// TIA Portal V18 export
ORGANIZATION_BLOCK "Main"   // OB1, LAD, ProgramCycle
TITLE = "Main Program Sweep (Cycle)"
{ S7_Optimized_Access := 'TRUE' }
VERSION : 0.1
// stored: AutoNumber true, IsIECCheckEnabled false, SetENOAutomatically false
   VAR_INPUT
      Initial_Call : Bool;   // Initial call of this OB
      Remanence : Bool;   // =True, if remanent data are available
   END_VAR
BEGIN

REGION Network 2
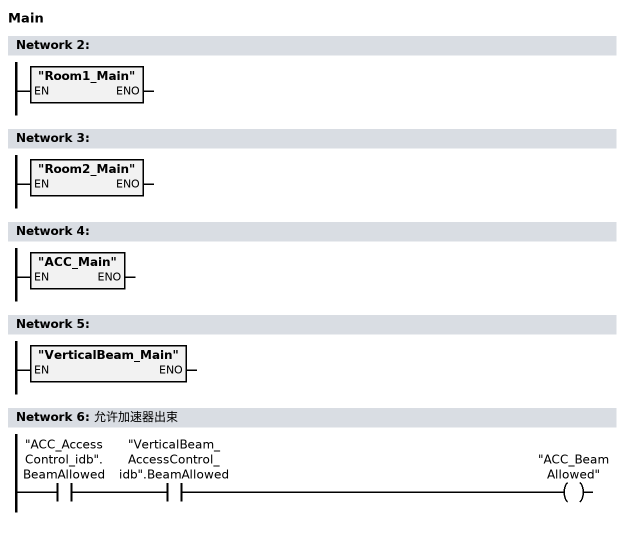
   RUNG wire#powerrail
      "Room1_Main"()
   END_RUNG
   // the same network as SCL:
   "Room1_Main"();
END_REGION

REGION Network 3
   RUNG wire#powerrail
      "Room2_Main"()
   END_RUNG
   // the same network as SCL:
   "Room2_Main"();
END_REGION

REGION Network 4
   RUNG wire#powerrail
      "ACC_Main"()
   END_RUNG
   // the same network as SCL:
   "ACC_Main"();
END_REGION

REGION Network 5
   RUNG wire#powerrail
      "VerticalBeam_Main"()
   END_RUNG
   // the same network as SCL:
   "VerticalBeam_Main"();
END_REGION

REGION Network 6: 允许加速器出束
   RUNG wire#powerrail
      Contact( "ACC_AccessControl_idb".BeamAllowed )
      Contact( "VerticalBeam_AccessControl_idb".BeamAllowed )
      Coil( "ACC_BeamAllowed" )
   END_RUNG
   // the same network as SCL:
   "ACC_BeamAllowed" := "ACC_AccessControl_idb".BeamAllowed AND "VerticalBeam_AccessControl_idb".BeamAllowed;
END_REGION
END_ORGANIZATION_BLOCK
